FUNCTION_BLOCK EliteBoard (* Service Interface Function Block Type *)
  (* Standard: 61499-2; Description: Copyright (c) 2021, 2022 Jonathan Lainer This program and the accompanying materials are made available under the terms of the Eclipse Public License 2.0 which is available at https://www.eclipse.org/legal/epl-2.0/ SPDX-License-Identifier: EPL-2.0 *)
  (* Version 1.0, 2021-02-22, Jonathan Lainer, Initial Contribution *)
  (* Version 3.0, 2025-04-14, Patrick Aigner, changed package *)
  PACKAGE eclipse4diac::io::eliteboard;
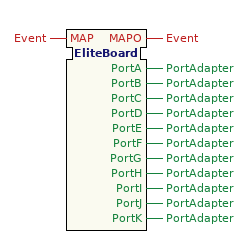
  EVENT_INPUT
    MAP;
  END_EVENT
  EVENT_OUTPUT
    MAPO;
  END_EVENT
  PLUGS
    PortA : eclipse4diac::io::eliteboard::PortAdapter;
    PortB : eclipse4diac::io::eliteboard::PortAdapter;
    PortC : eclipse4diac::io::eliteboard::PortAdapter;
    PortD : eclipse4diac::io::eliteboard::PortAdapter;
    PortE : eclipse4diac::io::eliteboard::PortAdapter;
    PortF : eclipse4diac::io::eliteboard::PortAdapter;
    PortG : eclipse4diac::io::eliteboard::PortAdapter;
    PortH : eclipse4diac::io::eliteboard::PortAdapter;
    PortI : eclipse4diac::io::eliteboard::PortAdapter;
    PortJ : eclipse4diac::io::eliteboard::PortAdapter;
    PortK : eclipse4diac::io::eliteboard::PortAdapter;
  END_PLUGS
END_FUNCTION_BLOCK
